INTERFACE I_HostNodes

PROPERTY Nodes : I_Nodes
GET
END_GET
END_PROPERTY

END_INTERFACE

(* stored: Version 1.1.0.1, ProductVersion 3.1.4024.12
   Itf I_HostNodes: Id {7df61bc8-9e76-43d8-902c-1f4a3879191e}
   Property Nodes: Id {fab13836-ac03-442d-82ab-adc0634fa43e}
   Get Get: Id {7aa44a45-2529-48b7-9d3c-afff5b216e3a} *)
